Universal Robots URScript: canpickerclient.script

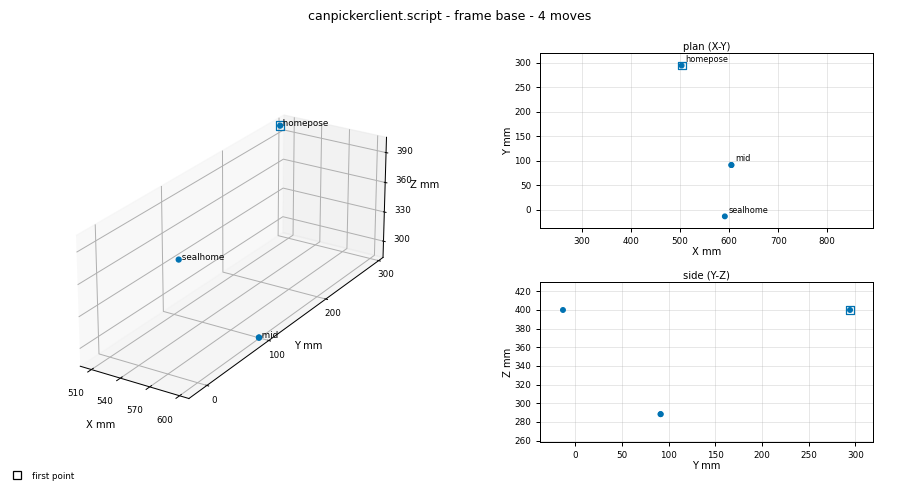
[picture p0: tool path of canpickerclient.script in frame base, 4 of 32 moves have a stored position in this frame; points joined in program order, loops and branches not executed]
def canpickerclient():
  set_tool_voltage(24)
  set_safety_mode_transition_hardness(1)
  set_gravity([0.0, 0.0, 9.82])
  step_count_2416d649_9ece_4dc5_960d_74b3799aade6 = 0.0
  thread Step_Counter_Thread_93d63abe_5f22_456b_b5e5_ea3f51299719():
    while (True):
      step_count_2416d649_9ece_4dc5_960d_74b3799aade6 = step_count_2416d649_9ece_4dc5_960d_74b3799aade6 + 1.0
      sync()
    end
  end
  run Step_Counter_Thread_93d63abe_5f22_456b_b5e5_ea3f51299719()
  set_standard_analog_input_domain(0, 1)
  set_standard_analog_input_domain(1, 1)
  set_tool_analog_input_domain(0, 1)
  set_tool_analog_input_domain(1, 1)
  set_analog_outputdomain(0, 0)
  set_analog_outputdomain(1, 0)
  set_input_actions_to_default()
  set_runstate_standard_digital_output_to_value(7, 2)
  set_tcp(p[0.0,0.0,0.0,0.0,0.0,0.0])
  set_payload(0.5)
  # begin: URCap Installation Node
  #   Source: External Control, 1.0.1, FZI Research Center for Information Technology
  #   Type: External Control
  # end: URCap Installation Node
  # begin: URCap Installation Node
  #   Source: RG - On Robot, 1.10.1, OnRobot A/S
  #   Type: RG Configuration
  global measure_width=0
  global grip_detected=False
  global lost_grip=False
  global zsysx=0
  global zsysy=0
  global zsysz=0.10205
  global zsysm=1.085
  global zmasx=0
  global zmasy=0
  global zmasz=0.23434
  global zslax=0
  global zslay=0
  global zslaz=0
  global zmasm=0
  global zslam=0
  global zslatcp=p[0,0,0,0,0,0]
  global zmastcp=p[0,0,0.23435,0,-0,-3.14159]
  thread lost_grip_thread():
  while True:
  set_tool_voltage(24)
  	if True ==get_digital_in(9):
  		sleep(0.024)
  		if True == grip_detected:
  			if False == get_digital_in(8):
  				grip_detected=False
  				lost_grip=True
  			end
  		end
  	set_tool_analog_input_domain(0, 1)
  	set_tool_analog_input_domain(1, 1)
  	zscale = (get_analog_in(2)-0.026)/2.9760034
  	zangle = zscale*1.57079633+-0.09424778
  	zwidth = 8.4+160*sin(zangle)
  	global measure_width = (floor(zwidth*10))/10-9.2
  	end
  	sync()
  end
  end
  lg_thr = run lost_grip_thread()
  def RG6(target_width=160, target_force=120, payload=0.0, set_payload=False, depth_compensation=False, slave=False):
  	set_tcp(p[0,0,0.23435,0,-0,-3.14159])
  	grip_detected=False
  	if slave:
  		slave_grip_detected=False
  	else:
  		master_grip_detected=False
  	end
  	timeout = 0
  	timeout_limit = 1250000
  	while get_digital_in(9) == False:
  	  if timeout > timeout_limit:
  	    break
  	  end
  	  timeout = timeout+1
  	  sync()
  	end
  	def bit(input):
  	  msb=65536
  	  local i=0
  	  local output=0
  	  while i<17:
  	    set_digital_out(8,True)
  	    if input>=msb:
  	      input=input-msb
  	      set_digital_out(9,False)
  	    else:
  	      set_digital_out(9,True)
  	    end
  	    if get_digital_in(8):
  	      out=1
  	    end
  	    sync()
  	    set_digital_out(8,False)
  	    sync()
  	    input=input*2
  	    output=output*2
  	    i=i+1
  	  end
  	  return output
  	end
  	target_width=target_width+9.2
  	if target_force>120:
  	target_force=120
  	end
  	if target_force<25:
  	target_force=25
  	end
  	if target_width>160:
  	target_width=160
  	end
  	if target_width<0:
  	target_width=0
  	end
  	rg_data=floor(target_width)*4
  	rg_data=rg_data+floor(target_force/5)*4*161
  	rg_data=rg_data+32768
  	if slave:
  	rg_data=rg_data+16384
  	end
  	bit(rg_data)
  	if slave==False:
  	t_w_rg=pose_trans(get_actual_tool_flange_pose(), zmastcp)
  	end
  	if slave:
  	t_w_rg=pose_trans(get_actual_tool_flange_pose(), zslatcp)
  	end
  	t_rg_w=pose_inv(t_w_rg)
  	if depth_compensation:
  	finger_length = 80.0/1000
  	finger_heigth_disp = 6.3/1000
  	center_displacement = 10.5/1000

  	start_pose = get_forward_kin()
  	set_analog_inputrange(2, 1)
  	zscale = (get_analog_in(2)-0.026)/2.9760034
  	zangle = zscale*1.57079633+-0.09424778
  	zwidth = 8.4+160*sin(zangle)

  	start_depth = cos(zangle)*finger_length

  	sleep(0.016)
  	timeout = 0
  	while get_digital_in(9) == True:
  	  timeout=timeout+1
  	  sleep(0.008)
  	  if timeout > 20:
  	    break
  	  end
  	end
  	timeout = 0
  	timeout_limit = 1250000
  	compensation_depth = 0
  	while get_digital_in(9) == False:
  	  zscale = (get_analog_in(2)-0.026)/2.9760034
  	  zangle = zscale*1.57079633+-0.09424778
  	  zwidth = 8.4+160*sin(zangle)
  	  measure_depth = cos(zangle)*finger_length
  	  compensation_depth = (measure_depth - start_depth)
  	  target_pose =pose_add(start_pose,pose_trans(pose_trans(t_w_rg, p[0,0,-compensation_depth,0,0,0]),t_rg_w))

  	  if timeout > timeout_limit:
  	    break
  	  end
  	  timeout=timeout+1
  	#  servoj(get_inverse_kin(target_pose), t=0.008, lookahead_time=0.033, gain=1500)
  	#  textmsg(point_dist(target_pose, get_forward_kin()))
  	#end
  	#textmsg("end gripper move!!!!!")
  	#nspeedthr = 0.001
  	#nspeed = norm(get_actual_tcp_speed())
  	#while nspeed > nspeedthr:
  	#  servoj(get_inverse_kin(target_pose), t=0.008, lookahead_time=0.033, gain=1500)
  	#  nspeed = norm(get_actual_tcp_speed())
  	#  textmsg(point_dist(target_pose, get_forward_kin()))
  	#end
  	servoj(get_inverse_kin(target_pose),0,0,0.008,0.01,2000)
  	if point_dist(target_pose, get_forward_kin()) > 0.005:
  	popup("Lower grasping force or max width",title="RG-lag threshold exceeded", warning=False, error=False, blocking=False)
  	end
  	end
  	act_comp_pose = p[0,0,0,0,0,0]
  	while norm(act_comp_pose) < norm(compensation_depth)-0.0002:
  	servoj(get_inverse_kin(target_pose),0,0,0.008,0.01,2000)
  	act_comp_pose = pose_trans(pose_inv(start_pose),get_forward_kin())
  	end
  	stopj(2)
  	end
  	if depth_compensation==False:
  	timeout = 0
  	timeout_count=20*0.008/0.008
  	while get_digital_in(9) == True:
  	  timeout = timeout+1
  	  sync()
  	  if timeout > timeout_count:
  	    break
  	  end
  	end
  	timeout = 0
  	timeout_limit = 1250000
  	while get_digital_in(9) == False:
  	  timeout = timeout+1
  	  sync()
  	  if timeout > timeout_limit:
  	    break
  	  end
  	end
  	end
  	sleep(0.024)
  	if set_payload:
  	if slave:
  	if get_analog_in(3)/0.5952007 < 1.42:
  	zslam=0
  	else:
  	zslam=payload
  	end
  	else:
  	if get_digital_in(8) == False:
  	zmasm=0
  	else:
  	zmasm=payload
  	end
  	end
  	zload=zmasm+zslam+zsysm
  	set_payload(zload,[(zsysx*zsysm+zmasx*zmasm+zslax*zslam)/zload,(zsysy*zsysm+zmasy*zmasm+zslay*zslam)/zload,(zsysz*zsysm+zmasz*zmasm+zslaz*zslam)/zload])
  	end
  	master_grip_detected=False
  	master_lost_grip=False
  	slave_grip_detected=False
  	slave_lost_grip=False
  	if True == get_digital_in(8):
  		master_grip_detected=True
  	end
  	if get_analog_in(3)/0.5952007>1.97:
  		slave_grip_detected=True
  	end
  	grip_detected=False
  	lost_grip=False
  	if True == get_digital_in(8):
  		grip_detected=True
  	end
  	zscale = (get_analog_in(2)-0.026)/2.9760034
  	zangle = zscale*1.57079633+-0.09424778
  	zwidth = 8.4+160*sin(zangle)
  	global measure_width = (floor(zwidth*10))/10-9.2
  	if slave:
  	slave_measure_width=measure_width
  	else:
  	master_measure_width=measure_width
  	end
  	return grip_detected
  end
  set_tool_voltage(24)
  set_tcp(p[0,0,0.23435,0,-0,-3.14159])
  # end: URCap Installation Node
  $ 1 "BeforeStart"
  $ 2 "rpicon≔rpc_factory('xmlrpc','http://192.168.1.100:50001')"
  global rpicon=rpc_factory("xmlrpc","http://192.168.1.100:50001")
  while (True):
    $ 3 "Robot Program"
    $ 4 "mid≔Point_4_const"
    global mid=p[0.6045247785102772,0.0914069590371725,0.28837445612697354,1.4953341567314073,2.4998807198840662,-1.0446828250517395]
    $ 5 "Loop"
    while (True):
      $ 6 "MoveJ"
      # begin: URCap Program Node
      #   Source: RG - On Robot, 1.10.1, OnRobot A/S
      #   Type: RG6
      $ 7 "RG6(20)"
      RG6(20,50,0.0,True,False,False)
      # end: URCap Program Node
      $ 8 "homepose" "breakAfter"
      movej(get_inverse_kin(p[.503078372310, .294269414884, .399963450268, -1.443377901300, -2.766126107933, .005980751993], qnear=[0.7848802208900452, -1.3780034224139612, -1.7669857184039515, -1.575134579335348, 1.586999773979187, 0.19088362157344818]), a=1.3962634015954636, v=1.0471975511965976)
      $ 9 "TinAvailable≔ False "
      global TinAvailable=  False
      $ 10 "Loop TinAvailable== False "
      while (TinAvailable==  False  ):
        $ 11 "TinAvailable≔rpicon.requestIsEmptyTin()"
        global TinAvailable=rpicon.requestIsEmptyTin()
      end
      $ 12 "TinTopPose≔rpicon.requestEmptyTinTopPose()"
      global TinTopPose=rpicon.requestEmptyTinTopPose()
      $ 13 "MoveJ"
      $ 14 "TinTopPose" "breakAfter"
      movej(TinTopPose, a=1.3962634015954636, v=1.0471975511965976)
      # begin: URCap Program Node
      #   Source: RG - On Robot, 1.10.1, OnRobot A/S
      #   Type: RG6
      $ 15 "RG6(120)"
      RG6(120,120,0.0,True,False,False)
      # end: URCap Program Node
      $ 16 "JointAngles≔rpicon.requestGripperRotationJointAngles(get_target_joint_positions(), 0)"
      global JointAngles=rpicon.requestGripperRotationJointAngles( get_target_joint_positions (), 0)
      $ 17 "RotatedPose≔get_forward_kin(JointAngles)"
      global RotatedPose=get_forward_kin(JointAngles)
      $ 18 "MoveJ"
      $ 19 "RotatedPose" "breakAfter"
      movej(RotatedPose, a=1.3962634015954636, v=1.0471975511965976)
      $ 20 "TinScanPose≔rpicon.requestEmptyTinScanPose(RotatedPose)"
      global TinScanPose=rpicon.requestEmptyTinScanPose(RotatedPose)
      $ 21 "MoveL"
      $ 22 "TinScanPose" "breakAfter"
      movel(pose_trans(p[0.0,0.0,0.0,0.0,0.0,0.0], TinScanPose), a=1.2, v=0.25)
      $ 23 "RfidVal≔rpicon.requestRFIDValidation()"
      global RfidVal=rpicon.requestRFIDValidation()
      $ 24 "If RfidVal == False "
      if (RfidVal ==  False  ):
        $ 25 "MoveL"
        $ 26 "RotatedPose" "breakAfter"
        movel(pose_trans(p[0.0,0.0,0.0,0.0,0.0,0.0], RotatedPose), a=1.2, v=0.25)
        $ 27 "JointAngles≔rpicon.requestGripperRotationJointAngles(get_target_joint_positions(), -179)"
        global JointAngles=rpicon.requestGripperRotationJointAngles( get_target_joint_positions (), -179)
        $ 28 "RotatedPose≔get_forward_kin(JointAngles)"
        global RotatedPose=get_forward_kin(JointAngles)
        $ 29 "MoveJ"
        $ 30 "RotatedPose" "breakAfter"
        movej(RotatedPose, a=1.3962634015954636, v=1.0471975511965976)
        $ 31 "TinScanPose≔rpicon.requestEmptyTinScanPose(RotatedPose)"
        global TinScanPose=rpicon.requestEmptyTinScanPose(RotatedPose)
        $ 32 "MoveL"
        $ 33 "TinScanPose" "breakAfter"
        movel(pose_trans(p[0.0,0.0,0.0,0.0,0.0,0.0], TinScanPose), a=1.2, v=0.25)
        $ 34 "Wait: 3.0"
        sleep(3.0)
        $ 35 "TinGrabPose≔rpicon.requestEmptyTinGrabPose(RotatedPose)"
        global TinGrabPose=rpicon.requestEmptyTinGrabPose(RotatedPose)
        $ 36 "MoveL"
        $ 37 "TinGrabPose" "breakAfter"
        movel(pose_trans(p[0.0,0.0,0.0,0.0,0.0,0.0], TinGrabPose), a=1.2, v=0.25)
        $ 38 "Wait: 3.0"
        sleep(3.0)
      end
      $ 39 "TinGrabPose≔rpicon.requestEmptyTinGrabPose(RotatedPose)"
      global TinGrabPose=rpicon.requestEmptyTinGrabPose(RotatedPose)
      $ 40 "MoveL"
      $ 41 "TinGrabPose" "breakAfter"
      movel(pose_trans(p[0.0,0.0,0.0,0.0,0.0,0.0], TinGrabPose), a=1.2, v=0.25)
      $ 42 "Wait: 3.0"
      sleep(3.0)
      # begin: URCap Program Node
      #   Source: RG - On Robot, 1.10.1, OnRobot A/S
      #   Type: RG6
      $ 43 "RG6(50)"
      RG6(50,50,0.0,True,False,False)
      # end: URCap Program Node
      $ 44 "TinLeavePose≔rpicon.requestEmptyTinLeavePose(TinGrabPose)"
      global TinLeavePose=rpicon.requestEmptyTinLeavePose(TinGrabPose)
      $ 45 "MoveL"
      $ 46 "TinLeavePose" "breakAfter"
      movel(pose_trans(p[0.0,0.0,0.0,0.0,0.0,0.0], TinLeavePose), a=1.2, v=0.25)
      $ 47 "If RfidVal== True "
      if (RfidVal==  True  ):
        $ 48 "MoveJ"
        $ 49 "mid" "breakAfter"
        movej(mid, a=1.3962634015954636, v=1.0471975511965976)
        $ 50 "CaningTopPose≔rpicon.requestCaningTopPose()"
        global CaningTopPose=rpicon.requestCaningTopPose()
        $ 51 "MoveJ"
        $ 52 "CaningTopPose" "breakAfter"
        movej(CaningTopPose, a=1.3962634015954636, v=1.0471975511965976)
        $ 53 "CaningGrabPose≔rpicon.requestCaningGrabPose(CaningTopPose)"
        global CaningGrabPose=rpicon.requestCaningGrabPose(CaningTopPose)
        $ 54 "MoveL"
        $ 55 "CaningGrabPose" "breakAfter"
        movel(pose_trans(p[0.0,0.0,0.0,0.0,0.0,0.0], CaningGrabPose), a=1.2, v=0.25)
        # begin: URCap Program Node
        #   Source: RG - On Robot, 1.10.1, OnRobot A/S
        #   Type: RG6
        $ 56 "RG6(120)"
        RG6(120,50,0.0,True,False,False)
        # end: URCap Program Node
        $ 57 "MoveL"
        $ 58 "CaningTopPose" "breakAfter"
        movel(pose_trans(p[0.0,0.0,0.0,0.0,0.0,0.0], CaningTopPose), a=1.2, v=0.25)
        $ 59 "Wait: 3.0"
        sleep(3.0)
        $ 60 "sealhome≔Point_5_const"
        global sealhome=p[0.5911775501945569,-0.013182414109391093,0.3999504844666265,-1.2566801328675798,1.1729687116978247,-1.2432864895180045]
        $ 61 "MoveL"
        $ 62 "sealhome" "breakAfter"
        movel(pose_trans(p[0.0,0.0,0.0,0.0,0.0,0.0], sealhome), a=1.2, v=0.25)
        $ 63 "Wait: 3.0"
        sleep(3.0)
        $ 64 "Wait: 3.0"
        sleep(3.0)
        $ 65 "SealVal≔rpicon.requestSealValidation()"
        global SealVal=rpicon.requestSealValidation()
        $ 68 "MoveJ"
        $ 69 "CaningGrabPose" "breakAfter"
        movej(CaningGrabPose, a=1.3962634015954636, v=1.0471975511965976)
        $ 70 "Wait: 3.0"
        sleep(3.0)
        $ 71 "CaningScanPose≔rpicon.requestCaningScanPose(CaningGrabPose)"
        global CaningScanPose=rpicon.requestCaningScanPose(CaningGrabPose)
        $ 72 "MoveL"
        $ 73 "CaningScanPose" "breakAfter"
        movel(pose_trans(p[0.0,0.0,0.0,0.0,0.0,0.0], CaningScanPose), a=1.2, v=0.25)
        $ 74 "Wait: 3.0"
        sleep(3.0)
        $ 75 "RfidUpdate≔rpicon.requestIsTinUpdated(SealVal)"
        global RfidUpdate=rpicon.requestIsTinUpdated(SealVal)
        $ 76 "Wait: 3.0"
        sleep(3.0)
        $ 77 "MoveL"
        $ 78 "CaningGrabPose" "breakAfter"
        movel(pose_trans(p[0.0,0.0,0.0,0.0,0.0,0.0], CaningGrabPose), a=1.2, v=0.25)
        $ 79 "Wait: 3.0"
        sleep(3.0)
        # begin: URCap Program Node
        #   Source: RG - On Robot, 1.10.1, OnRobot A/S
        #   Type: RG6
        $ 80 "RG6(50)"
        RG6(50,50,0.0,True,False,False)
        # end: URCap Program Node
        $ 81 "MoveL"
        $ 82 "CaningTopPose" "breakAfter"
        movel(pose_trans(p[0.0,0.0,0.0,0.0,0.0,0.0], CaningTopPose), a=1.2, v=0.25)
        $ 83 "If SealVal== True  and  RfidUpdate== True "
        if (SealVal==  True    and   RfidUpdate==  True  ):
          $ 84 "pvTopNextPose≔rpicon.requestPackingValidTopNextPose()"
          global pvTopNextPose=rpicon.requestPackingValidTopNextPose()
          $ 85 "MoveJ"
          $ 86 "pvTopNextPose" "breakAfter"
          movej(pvTopNextPose, a=1.3962634015954636, v=1.0471975511965976)
          $ 87 "pvRelNextPose≔rpicon.requestPackingValidReleaseNextPose(pvTopNextPose)"
          global pvRelNextPose=rpicon.requestPackingValidReleaseNextPose(pvTopNextPose)
          $ 88 "MoveL"
          $ 89 "pvRelNextPose" "breakAfter"
          movel(pose_trans(p[0.0,0.0,0.0,0.0,0.0,0.0], pvRelNextPose), a=1.2, v=0.25)
          # begin: URCap Program Node
          #   Source: RG - On Robot, 1.10.1, OnRobot A/S
          #   Type: RG6
          $ 90 "RG6(120)"
          RG6(120,50,0.0,True,False,False)
          # end: URCap Program Node
          $ 91 "MoveL"
          $ 92 "pvTopNextPose" "breakAfter"
          movel(pose_trans(p[0.0,0.0,0.0,0.0,0.0,0.0], pvTopNextPose), a=1.2, v=0.25)
        else:
          $ 93 "Else" "noBreak"
          $ 94 "pnvTopNextPose≔rpicon.requestPackingNotValidTopNextPose()"
          global pnvTopNextPose=rpicon.requestPackingNotValidTopNextPose()
          $ 95 "MoveJ"
          $ 96 "pnvTopNextPose" "breakAfter"
          movej(pnvTopNextPose, a=1.3962634015954636, v=1.0471975511965976)
          $ 97 "pnvRelNextPose≔rpicon.requestPackingNotValidReleaseNextPose(pnvTopNextPose)"
          global pnvRelNextPose=rpicon.requestPackingNotValidReleaseNextPose(pnvTopNextPose)
          $ 98 "MoveL"
          $ 99 "pnvRelNextPose" "breakAfter"
          movel(pose_trans(p[0.0,0.0,0.0,0.0,0.0,0.0], pnvRelNextPose), a=1.2, v=0.25)
          # begin: URCap Program Node
          #   Source: RG - On Robot, 1.10.1, OnRobot A/S
          #   Type: RG6
          $ 100 "RG6(120)"
          RG6(120,50,0.0,True,False,False)
          # end: URCap Program Node
          $ 101 "MoveL"
          $ 102 "pnvTopNextPose" "breakAfter"
          movel(pose_trans(p[0.0,0.0,0.0,0.0,0.0,0.0], pnvTopNextPose), a=1.2, v=0.25)
        end
      else:
        $ 103 "Else" "noBreak"
        $ 104 "CaningTopPose≔rpicon.requestCaningTopPose()"
        global CaningTopPose=rpicon.requestCaningTopPose()
        $ 105 "MoveJ"
        $ 106 "mid" "breakAfter"
        movej(mid, a=1.3962634015954636, v=1.0471975511965976)
        $ 107 "MoveJ"
        $ 108 "CaningTopPose" "breakAfter"
        movej(CaningTopPose, a=1.3962634015954636, v=1.0471975511965976)
        $ 109 "pnvTopNextPose≔rpicon.requestPackingNotValidTopNextPose()"
        global pnvTopNextPose=rpicon.requestPackingNotValidTopNextPose()
        $ 110 "MoveJ"
        $ 111 "pnvTopNextPose" "breakAfter"
        movej(pnvTopNextPose, a=1.3962634015954636, v=1.0471975511965976)
        $ 112 "pnvRelNextPose≔rpicon.requestPackingNotValidReleaseNextPose(pnvTopNextPose)"
        global pnvRelNextPose=rpicon.requestPackingNotValidReleaseNextPose(pnvTopNextPose)
        $ 113 "MoveL"
        $ 114 "pnvRelNextPose" "breakAfter"
        movel(pose_trans(p[0.0,0.0,0.0,0.0,0.0,0.0], pnvRelNextPose), a=1.2, v=0.25)
        $ 115 "Wait: 3.0"
        sleep(3.0)
        # begin: URCap Program Node
        #   Source: RG - On Robot, 1.10.1, OnRobot A/S
        #   Type: RG6
        $ 116 "RG6(120)"
        RG6(120,50,0.0,True,False,False)
        # end: URCap Program Node
        $ 117 "MoveL"
        $ 118 "pnvTopNextPose" "breakAfter"
        movel(pose_trans(p[0.0,0.0,0.0,0.0,0.0,0.0], pnvTopNextPose), a=1.2, v=0.25)
      end
    end
  end
end
